// TIA Portal project "OpcUaClient" (V15.1)

(* hardware
DEVICE "S71500/ET200MP-Station_1"  S7-1500 station
   slot 0: "Profilschiene_0"  Rack  6ES7 590-1***0-0AA0
   slot 1: "PLC"  CPU 1513F-1 PN  6ES7 513-1FL02-0AB0  V2.6
      slot 3: "CPU-Display_1"  6ES7591-1AA00-0AA0
*)

// ===== PLC "PLC"  CPU 1513F-1 PN =====

VAR_GLOBAL   // PLC tag table "Standard-Variablentabelle"
   "System_Byte" AT %MB1 : Byte;
   "FirstScan" AT %M1.0 : Bool;
   "DiagStatusUpdate" AT %M1.1 : Bool;
   "AlwaysTRUE" AT %M1.2 : Bool;
   "AlwaysFALSE" AT %M1.3 : Bool;
   "Clock_Byte" AT %MB0 : Byte;
   "Clock_10Hz" AT %M0.0 : Bool;
   "Clock_5Hz" AT %M0.1 : Bool;
   "Clock_2.5Hz" AT %M0.2 : Bool;
   "Clock_2Hz" AT %M0.3 : Bool;
   "Clock_1.25Hz" AT %M0.4 : Bool;
   "Clock_1Hz" AT %M0.5 : Bool;
   "Clock_0.625Hz" AT %M0.6 : Bool;
   "Clock_0.5Hz" AT %M0.7 : Bool;
   "Tag_1" AT %M100.0 : Bool;
   "Tag_2" AT %M300.0 : Bool;
   "Tag_3" AT %M300.1 : Bool;
   "Tag_4" AT %MD310 : DWord;
   "Tag_5" AT %M300.2 : Bool;
   "Tag_6" AT %M200.0 : Bool;
   "Tag_7" AT %M200.2 : Bool;
   "Tag_8" AT %MD210 : DWord;
   "Tag_9" AT %M200.1 : Bool;
   "Tag_10" AT %M600.0 : Bool;
   "Tag_11" AT %M400.0 : Bool;
   "Tag_12" AT %M1000.0 : Bool;
   "Tag_13" AT %M1000.1 : Bool;
   "Tag_14" AT %M1000.2 : Bool;
   "Tag_15" AT %M1000.3 : Bool;
   "Tag_16" AT %M1000.4 : Bool;
   "Tag_17" AT %M1000.5 : Bool;
END_VAR

VAR_GLOBAL CONSTANT   // PLC tag table "Tag table from XML_1"
   "OpcUa_Good" : DWord := 16#00000000;   // Everything is as expected.
   "OpcUa_Uncertain" : DWord := 16#40000000;   // Something unexpected occurred but the results still maybe useable.
   "OpcUa_Bad" : DWord := 16#80000000;   // An error occurred.
   "OpcUa_BadUnexpectedError" : DWord := 16#80010000;   // An unexpected error occurred.
   "OpcUa_BadInternalError" : DWord := 16#80020000;   // An internal error occurred as a result of a programming or configuration error.
   "OpcUa_BadOutOfMemory" : DWord := 16#80030000;   // Not enough memory to complete the operation.
   "OpcUa_BadResourceUnavailable" : DWord := 16#80040000;   // An operating system resource is not available.
   "OpcUa_BadCommunicationError" : DWord := 16#80050000;   // A low level communication error occurred.
   "OpcUa_BadEncodingError" : DWord := 16#80060000;   // Encoding halted because of invalid data in the objects being serialized.
   "OpcUa_BadDecodingError" : DWord := 16#80070000;   // Decoding halted because of invalid data in the stream.
   "OpcUa_BadEncodingLimitsExceeded" : DWord := 16#80080000;   // The message encoding/decoding limits imposed by the stack have been exceeded.
   "OpcUa_BadRequestTooLarge" : DWord := 16#80B80000;   // The request message size exceeds limits set by the server.
   "OpcUa_BadResponseTooLarge" : DWord := 16#80B90000;   // The response message size exceeds limits set by the client.
   "OpcUa_BadUnknownResponse" : DWord := 16#80090000;   // An unrecognized response was received from the server.
   "OpcUa_BadTimeout" : DWord := 16#800A0000;   // The operation timed out.
   "OpcUa_BadServiceUnsupported" : DWord := 16#800B0000;   // The server does not support the requested service.
   "OpcUa_BadShutdown" : DWord := 16#800C0000;   // The operation was cancelled because the application is shutting down.
   "OpcUa_BadServerNotConnected" : DWord := 16#800D0000;   // The operation could not complete because the client is not connected to the server.
   "OpcUa_BadServerHalted" : DWord := 16#800E0000;   // The server has stopped and cannot process any requests.
   "OpcUa_BadNothingToDo" : DWord := 16#800F0000;   // There was nothing to do because the client passed a list of operations with no elements.
   "OpcUa_BadTooManyOperations" : DWord := 16#80100000;   // The request could not be processed because it specified too many operations.
   "OpcUa_BadTooManyMonitoredItems" : DWord := 16#80DB0000;   // The request could not be processed because there are too many monitored items in the subscription.
   "OpcUa_BadDataTypeIdUnknown" : DWord := 16#80110000;   // The extension object cannot be (de)serialized because the data type id is not recognized.
   "OpcUa_BadCertificateInvalid" : DWord := 16#80120000;   // The certificate provided as a parameter is not valid.
   "OpcUa_BadSecurityChecksFailed" : DWord := 16#80130000;   // An error occurred verifying security.
   "OpcUa_BadCertificateTimeInvalid" : DWord := 16#80140000;   // The certificate has expired or is not yet valid.
   "OpcUa_BadCertificateIssuerTimeInvalid" : DWord := 16#80150000;   // An issuer certificate has expired or is not yet valid.
   "OpcUa_BadCertificateHostNameInvalid" : DWord := 16#80160000;   // The HostName used to connect to a server does not match a HostName in the certificate.
   "OpcUa_BadCertificateUriInvalid" : DWord := 16#80170000;   // The URI specified in the ApplicationDescription does not match the URI in the certificate.
   "OpcUa_BadCertificateUseNotAllowed" : DWord := 16#80180000;   // The certificate may not be used for the requested operation.
   "OpcUa_BadCertificateIssuerUseNotAllowed" : DWord := 16#80190000;   // The issuer certificate may not be used for the requested operation.
   "OpcUa_BadCertificateUntrusted" : DWord := 16#801A0000;   // The certificate is not trusted.
   "OpcUa_BadCertificateRevocationUnknown" : DWord := 16#801B0000;   // It was not possible to determine if the certificate has been revoked.
   "OpcUa_BadCertificateIssuerRevocationUnknown" : DWord := 16#801C0000;   // It was not possible to determine if the issuer certificate has been revoked.
   "OpcUa_BadCertificateRevoked" : DWord := 16#801D0000;   // The certificate has been revoked.
   "OpcUa_BadCertificateIssuerRevoked" : DWord := 16#801E0000;   // The issuer certificate has been revoked.
   "OpcUa_BadCertificateChainIncomplete" : DWord := 16#810D0000;   // The certificate chain is incomplete.
   "OpcUa_BadUserAccessDenied" : DWord := 16#801F0000;   // User does not have permission to perform the requested operation.
   "OpcUa_BadIdentityTokenInvalid" : DWord := 16#80200000;   // The user identity token is not valid.
   "OpcUa_BadIdentityTokenRejected" : DWord := 16#80210000;   // The user identity token is valid but the server has rejected it.
   "OpcUa_BadSecureChannelIdInvalid" : DWord := 16#80220000;   // The specified secure channel is no longer valid.
   "OpcUa_BadInvalidTimestamp" : DWord := 16#80230000;   // The timestamp is outside the range allowed by the server.
   "OpcUa_BadNonceInvalid" : DWord := 16#80240000;   // The nonce does appear to be not a random value or it is not the correct length.
   "OpcUa_BadSessionIdInvalid" : DWord := 16#80250000;   // The session id is not valid.
   "OpcUa_BadSessionClosed" : DWord := 16#80260000;   // The session was closed by the client.
   "OpcUa_BadSessionNotActivated" : DWord := 16#80270000;   // The session cannot be used because ActivateSession has not been called.
   "OpcUa_BadSubscriptionIdInvalid" : DWord := 16#80280000;   // The subscription id is not valid.
   "OpcUa_BadRequestHeaderInvalid" : DWord := 16#802A0000;   // The header for the request is missing or invalid.
   "OpcUa_BadTimestampsToReturnInvalid" : DWord := 16#802B0000;   // The timestamps to return parameter is invalid.
   "OpcUa_BadRequestCancelledByClient" : DWord := 16#802C0000;   // The request was cancelled by the client.
   "OpcUa_BadTooManyArguments" : DWord := 16#80E50000;   // Too many arguments were provided.
   "OpcUa_BadLicenseExpired" : DWord := 16#810E0000;   // The server requires a license to operate in general or to perform a service or operation, but existing license is expired.
   "OpcUa_BadLicenseLimitsExceeded" : DWord := 16#810F0000;   // The server has limits on number of allowed operations / objects, based on installed licenses, and these limits where exceeded.
   "OpcUa_BadLicenseNotAvailable" : DWord := 16#81100000;   // The server does not have a license which is required to operate in general or to perform a service or operation.
   "OpcUa_GoodSubscriptionTransferred" : DWord := 16#002D0000;   // The subscription was transferred to another session.
   "OpcUa_GoodCompletesAsynchronously" : DWord := 16#002E0000;   // The processing will complete asynchronously.
   "OpcUa_GoodOverload" : DWord := 16#002F0000;   // Sampling has slowed down due to resource limitations.
   "OpcUa_GoodClamped" : DWord := 16#00300000;   // The value written was accepted but was clamped.
   "OpcUa_BadNoCommunication" : DWord := 16#80310000;   // Communication with the data source is defined, but not established, and there is no last known value available.
   "OpcUa_BadWaitingForInitialData" : DWord := 16#80320000;   // Waiting for the server to obtain values from the underlying data source.
   "OpcUa_BadNodeIdInvalid" : DWord := 16#80330000;   // The syntax of the node id is not valid.
   "OpcUa_BadNodeIdUnknown" : DWord := 16#80340000;   // The node id refers to a node that does not exist in the server address space.
   "OpcUa_BadAttributeIdInvalid" : DWord := 16#80350000;   // The attribute is not supported for the specified Node.
   "OpcUa_BadIndexRangeInvalid" : DWord := 16#80360000;   // The syntax of the index range parameter is invalid.
   "OpcUa_BadIndexRangeNoData" : DWord := 16#80370000;   // No data exists within the range of indexes specified.
   "OpcUa_BadDataEncodingInvalid" : DWord := 16#80380000;   // The data encoding is invalid.
   "OpcUa_BadDataEncodingUnsupported" : DWord := 16#80390000;   // The server does not support the requested data encoding for the node.
   "OpcUa_BadNotReadable" : DWord := 16#803A0000;   // The access level does not allow reading or subscribing to the Node.
   "OpcUa_BadNotWritable" : DWord := 16#803B0000;   // The access level does not allow writing to the Node.
   "OpcUa_BadOutOfRange" : DWord := 16#803C0000;   // The value was out of range.
   "OpcUa_BadNotSupported" : DWord := 16#803D0000;   // The requested operation is not supported.
   "OpcUa_BadNotFound" : DWord := 16#803E0000;   // A requested item was not found or a search operation ended without success.
   "OpcUa_BadObjectDeleted" : DWord := 16#803F0000;   // The object cannot be used because it has been deleted.
   "OpcUa_BadNotImplemented" : DWord := 16#80400000;   // Requested operation is not implemented.
   "OpcUa_BadMonitoringModeInvalid" : DWord := 16#80410000;   // The monitoring mode is invalid.
   "OpcUa_BadMonitoredItemIdInvalid" : DWord := 16#80420000;   // The monitoring item id does not refer to a valid monitored item.
   "OpcUa_BadMonitoredItemFilterInvalid" : DWord := 16#80430000;   // The monitored item filter parameter is not valid.
   "OpcUa_BadMonitoredItemFilterUnsupported" : DWord := 16#80440000;   // The server does not support the requested monitored item filter.
   "OpcUa_BadFilterNotAllowed" : DWord := 16#80450000;   // A monitoring filter cannot be used in combination with the attribute specified.
   "OpcUa_BadStructureMissing" : DWord := 16#80460000;   // A mandatory structured parameter was missing or null.
   "OpcUa_BadEventFilterInvalid" : DWord := 16#80470000;   // The event filter is not valid.
   "OpcUa_BadContentFilterInvalid" : DWord := 16#80480000;   // The content filter is not valid.
   "OpcUa_BadFilterOperatorInvalid" : DWord := 16#80C10000;   // An unregognized operator was provided in a filter.
   "OpcUa_BadFilterOperatorUnsupported" : DWord := 16#80C20000;   // A valid operator was provided, but the server does not provide support for this filter operator.
   "OpcUa_BadFilterOperandCountMismatch" : DWord := 16#80C30000;   // The number of operands provided for the filter operator was less then expected for the operand provided.
   "OpcUa_BadFilterOperandInvalid" : DWord := 16#80490000;   // The operand used in a content filter is not valid.
   "OpcUa_BadFilterElementInvalid" : DWord := 16#80C40000;   // The referenced element is not a valid element in the content filter.
   "OpcUa_BadFilterLiteralInvalid" : DWord := 16#80C50000;   // The referenced literal is not a valid value.
   "OpcUa_BadContinuationPointInvalid" : DWord := 16#804A0000;   // The continuation point provide is longer valid.
   "OpcUa_BadNoContinuationPoints" : DWord := 16#804B0000;   // The operation could not be processed because all continuation points have been allocated.
   "OpcUa_BadReferenceTypeIdInvalid" : DWord := 16#804C0000;   // The operation could not be processed because all continuation points have been allocated.
   "OpcUa_BadBrowseDirectionInvalid" : DWord := 16#804D0000;   // The browse direction is not valid.
   "OpcUa_BadNodeNotInView" : DWord := 16#804E0000;   // The node is not part of the view.
   "OpcUa_BadNumericOverflow" : DWord := 16#81120000;   // The number was not accepted because of a numeric overflow.
   "OpcUa_BadServerUriInvalid" : DWord := 16#804F0000;   // The ServerUri is not a valid URI.
   "OpcUa_BadServerNameMissing" : DWord := 16#80500000;   // No ServerName was specified.
   "OpcUa_BadDiscoveryUrlMissing" : DWord := 16#80510000;   // No DiscoveryUrl was specified.
   "OpcUa_BadSempahoreFileMissing" : DWord := 16#80520000;   // The semaphore file specified by the client is not valid.
   "OpcUa_BadRequestTypeInvalid" : DWord := 16#80530000;   // The security token request type is not valid.
   "OpcUa_BadSecurityModeRejected" : DWord := 16#80540000;   // The security mode does not meet the requirements set by the server.
   "OpcUa_BadSecurityPolicyRejected" : DWord := 16#80550000;   // The security policy does not meet the requirements set by the server.
   "OpcUa_BadTooManySessions" : DWord := 16#80560000;   // The server has reached its maximum number of sessions.
   "OpcUa_BadUserSignatureInvalid" : DWord := 16#80570000;   // The user token signature is missing or invalid.
   "OpcUa_BadApplicationSignatureInvalid" : DWord := 16#80580000;   // The signature generated with the client certificate is missing or invalid.
   "OpcUa_BadNoValidCertificates" : DWord := 16#80590000;   // The client did not provide at least one software certificate that is valid and meets the profile requirements for the server.
   "OpcUa_BadIdentityChangeNotSupported" : DWord := 16#80C60000;   // The server does not support changing the user identity assigned to the session.
   "OpcUa_BadRequestCancelledByRequest" : DWord := 16#805A0000;   // The request was cancelled by the client with the Cancel service.
   "OpcUa_BadParentNodeIdInvalid" : DWord := 16#805B0000;   // The parent node id does not to refer to a valid node.
   "OpcUa_BadReferenceNotAllowed" : DWord := 16#805C0000;   // The reference could not be created because it violates constraints imposed by the data model.
   "OpcUa_BadNodeIdRejected" : DWord := 16#805D0000;   // The requested node id was reject because it was either invalid or server does not allow node ids to be specified by the client.
   "OpcUa_BadNodeIdExists" : DWord := 16#805E0000;   // The requested node id is already used by another node.
   "OpcUa_BadNodeClassInvalid" : DWord := 16#805F0000;   // The node class is not valid.
   "OpcUa_BadBrowseNameInvalid" : DWord := 16#80600000;   // The browse name is invalid.
   "OpcUa_BadBrowseNameDuplicated" : DWord := 16#80610000;   // The browse name is not unique among nodes that share the same relationship with the parent.
   "OpcUa_BadNodeAttributesInvalid" : DWord := 16#80620000;   // The node attributes are not valid for the node class.
   "OpcUa_BadTypeDefinitionInvalid" : DWord := 16#80630000;   // The type definition node id does not reference an appropriate type node.
   "OpcUa_BadSourceNodeIdInvalid" : DWord := 16#80640000;   // The source node id does not reference a valid node.
   "OpcUa_BadTargetNodeIdInvalid" : DWord := 16#80650000;   // The target node id does not reference a valid node.
   "OpcUa_BadDuplicateReferenceNotAllowed" : DWord := 16#80660000;   // The reference type between the nodes is already defined.
   "OpcUa_BadInvalidSelfReference" : DWord := 16#80670000;   // The server does not allow this type of self reference on this node.
   "OpcUa_BadReferenceLocalOnly" : DWord := 16#80680000;   // The reference type is not valid for a reference to a remote server.
   "OpcUa_BadNoDeleteRights" : DWord := 16#80690000;   // The server will not allow the node to be deleted.
   "OpcUa_UncertainReferenceNotDeleted" : DWord := 16#40BC0000;   // The server was not able to delete all target references.
   "OpcUa_BadServerIndexInvalid" : DWord := 16#806A0000;   // The server index is not valid.
   "OpcUa_BadViewIdUnknown" : DWord := 16#806B0000;   // The view id does not refer to a valid view node.
   "OpcUa_BadViewTimestampInvalid" : DWord := 16#80C90000;   // The view timestamp is not available or not supported.
   "OpcUa_BadViewParameterMismatch" : DWord := 16#80CA0000;   // The view parameters are not consistent with each other.
   "OpcUa_BadViewVersionInvalid" : DWord := 16#80CB0000;   // The view version is not available or not supported.
   "OpcUa_UncertainNotAllNodesAvailable" : DWord := 16#40C00000;   // The list of references may not be complete because the underlying system is not available.
   "OpcUa_GoodResultsMayBeIncomplete" : DWord := 16#00BA0000;   // The server should have followed a reference to a node in a remote server but did not. The result set may be incomplete.
   "OpcUa_BadNotTypeDefinition" : DWord := 16#80C80000;   // The provided Nodeid was not a type definition nodeid.
   "OpcUa_UncertainReferenceOutOfServer" : DWord := 16#406C0000;   // One of the references to follow in the relative path references to a node in the address space in another server.
   "OpcUa_BadTooManyMatches" : DWord := 16#806D0000;   // The requested operation has too many matches to return.
   "OpcUa_BadQueryTooComplex" : DWord := 16#806E0000;   // The requested operation requires too many resources in the server.
   "OpcUa_BadNoMatch" : DWord := 16#806F0000;   // The requested operation has no match to return.
   "OpcUa_BadMaxAgeInvalid" : DWord := 16#80700000;   // The max age parameter is invalid.
   "OpcUa_BadSecurityModeInsufficient" : DWord := 16#80E60000;   // The operation is not permitted over the current secure channel.
   "OpcUa_BadHistoryOperationInvalid" : DWord := 16#80710000;   // The history details parameter is not valid.
   "OpcUa_BadHistoryOperationUnsupported" : DWord := 16#80720000;   // The server does not support the requested operation.
   "OpcUa_BadInvalidTimestampArgument" : DWord := 16#80BD0000;   // The defined timestamp to return was invalid.
   "OpcUa_BadWriteNotSupported" : DWord := 16#80730000;   // The server does not support writing the combination of value, status and timestamps provided.
   "OpcUa_BadTypeMismatch" : DWord := 16#80740000;   // The value supplied for the attribute is not of the same type as the attributes value.
   "OpcUa_BadMethodInvalid" : DWord := 16#80750000;   // The method id does not refer to a method for the specified object.
   "OpcUa_BadArgumentsMissing" : DWord := 16#80760000;   // The client did not specify all of the input arguments for the method.
   "OpcUa_BadNotExecutable" : DWord := 16#81110000;   // The executable attribute does not allow the execution of the method.
   "OpcUa_BadTooManySubscriptions" : DWord := 16#80770000;   // The server has reached its maximum number of subscriptions.
   "OpcUa_BadTooManyPublishRequests" : DWord := 16#80780000;   // The server has reached the maximum number of queued publish requests.
   "OpcUa_BadNoSubscription" : DWord := 16#80790000;   // There is no subscription available for this session.
   "OpcUa_BadSequenceNumberUnknown" : DWord := 16#807A0000;   // The sequence number is unknown to the server.
   "OpcUa_BadMessageNotAvailable" : DWord := 16#807B0000;   // The requested notification message is no longer available.
   "OpcUa_BadInsufficientClientProfile" : DWord := 16#807C0000;   // The client of the current session does not support one or more Profiles that are necessary for the subscription.
   "OpcUa_BadStateNotActive" : DWord := 16#80BF0000;   // The sub-state machine is not currently active.
   "OpcUa_BadTcpServerTooBusy" : DWord := 16#807D0000;   // The server cannot process the request because it is too busy.
   "OpcUa_BadTcpMessageTypeInvalid" : DWord := 16#807E0000;   // The type of the message specified in the header invalid.
   "OpcUa_BadTcpSecureChannelUnknown" : DWord := 16#807F0000;   // The SecureChannelId and/or TokenId are not currently in use.
   "OpcUa_BadTcpMessageTooLarge" : DWord := 16#80800000;   // The size of the message specified in the header is too large.
   "OpcUa_BadTcpNotEnoughResources" : DWord := 16#80810000;   // There are not enough resources to process the request.
   "OpcUa_BadTcpInternalError" : DWord := 16#80820000;   // An internal error occurred.
   "OpcUa_BadTcpEndpointUrlInvalid" : DWord := 16#80830000;   // The server does not recognize the QueryString specified.
   "OpcUa_BadRequestInterrupted" : DWord := 16#80840000;   // The request could not be sent because of a network interruption.
   "OpcUa_BadRequestTimeout" : DWord := 16#80850000;   // Timeout occurred while processing the request.
   "OpcUa_BadSecureChannelClosed" : DWord := 16#80860000;   // The secure channel has been closed.
   "OpcUa_BadSecureChannelTokenUnknown" : DWord := 16#80870000;   // The token has expired or is not recognized.
   "OpcUa_BadSequenceNumberInvalid" : DWord := 16#80880000;   // The sequence number is not valid.
   "OpcUa_BadProtocolVersionUnsupported" : DWord := 16#80BE0000;   // The applications do not have compatible protocol versions.
   "OpcUa_BadConfigurationError" : DWord := 16#80890000;   // There is a problem with the configuration that affects the usefulness of the value.
   "OpcUa_BadNotConnected" : DWord := 16#808A0000;   // The variable should receive its value from another variable, but has never been configured to do so.
   "OpcUa_BadDeviceFailure" : DWord := 16#808B0000;   // There has been a failure in the device/data source that generates the value that has affected the value.
   "OpcUa_BadSensorFailure" : DWord := 16#808C0000;   // There has been a failure in the sensor from which the value is derived by the device/data source.
   "OpcUa_BadOutOfService" : DWord := 16#808D0000;   // The source of the data is not operational.
   "OpcUa_BadDeadbandFilterInvalid" : DWord := 16#808E0000;   // The deadband filter is not valid.
   "OpcUa_UncertainNoCommunicationLastUsableValue" : DWord := 16#408F0000;   // Communication to the data source has failed. The variable value is the last value that had a good quality.
   "OpcUa_UncertainLastUsableValue" : DWord := 16#40900000;   // Whatever was updating this value has stopped doing so.
   "OpcUa_UncertainSubstituteValue" : DWord := 16#40910000;   // The value is an operational value that was manually overwritten.
   "OpcUa_UncertainInitialValue" : DWord := 16#40920000;   // The value is an initial value for a variable that normally receives its value from another variable.
   "OpcUa_UncertainSensorNotAccurate" : DWord := 16#40930000;   // The value is at one of the sensor limits.
   "OpcUa_UncertainEngineeringUnitsExceeded" : DWord := 16#40940000;   // The value is outside of the range of values defined for this parameter.
   "OpcUa_UncertainSubNormal" : DWord := 16#40950000;   // The value is derived from multiple sources and has less than the required number of Good sources.
   "OpcUa_GoodLocalOverride" : DWord := 16#00960000;   // The value has been overridden.
   "OpcUa_BadRefreshInProgress" : DWord := 16#80970000;   // This Condition refresh failed, a Condition refresh operation is already in progress.
   "OpcUa_BadConditionAlreadyDisabled" : DWord := 16#80980000;   // This condition has already been disabled.
   "OpcUa_BadConditionAlreadyEnabled" : DWord := 16#80CC0000;   // This condition has already been enabled.
   "OpcUa_BadConditionDisabled" : DWord := 16#80990000;   // Property not available, this condition is disabled.
   "OpcUa_BadEventIdUnknown" : DWord := 16#809A0000;   // The specified event id is not recognized.
   "OpcUa_BadEventNotAcknowledgeable" : DWord := 16#80BB0000;   // The event cannot be acknowledged.
   "OpcUa_BadDialogNotActive" : DWord := 16#80CD0000;   // The dialog condition is not active.
   "OpcUa_BadDialogResponseInvalid" : DWord := 16#80CE0000;   // The response is not valid for the dialog.
   "OpcUa_BadConditionBranchAlreadyAcked" : DWord := 16#80CF0000;   // The condition branch has already been acknowledged.
   "OpcUa_BadConditionBranchAlreadyConfirmed" : DWord := 16#80D00000;   // The condition branch has already been confirmed.
   "OpcUa_BadConditionAlreadyShelved" : DWord := 16#80D10000;   // The condition has already been shelved.
   "OpcUa_BadConditionNotShelved" : DWord := 16#80D20000;   // The condition is not currently shelved.
   "OpcUa_BadShelvingTimeOutOfRange" : DWord := 16#80D30000;   // The shelving time not within an acceptable range.
   "OpcUa_BadNoData" : DWord := 16#809B0000;   // No data exists for the requested time range or event filter.
   "OpcUa_BadBoundNotFound" : DWord := 16#80D70000;   // No data found to provide upper or lower bound value.
   "OpcUa_BadBoundNotSupported" : DWord := 16#80D80000;   // The server cannot retrieve a bound for the variable.
   "OpcUa_BadDataLost" : DWord := 16#809D0000;   // Data is missing due to collection started/stopped/lost.
   "OpcUa_BadDataUnavailable" : DWord := 16#809E0000;   // Expected data is unavailable for the requested time range due to an un-mounted volume, an off-line archive or tape, or similar reason for temporary unavailability.
   "OpcUa_BadEntryExists" : DWord := 16#809F0000;   // The data or event was not successfully inserted because a matching entry exists.
   "OpcUa_BadNoEntryExists" : DWord := 16#80A00000;   // The data or event was not successfully updated because no matching entry exists.
   "OpcUa_BadTimestampNotSupported" : DWord := 16#80A10000;   // The client requested history using a timestamp format the server does not support (i.e requested ServerTimestamp when server only supports SourceTimestamp).
   "OpcUa_GoodEntryInserted" : DWord := 16#00A20000;   // The data or event was successfully inserted into the historical database.
   "OpcUa_GoodEntryReplaced" : DWord := 16#00A30000;   // The data or event field was successfully replaced in the historical database.
   "OpcUa_UncertainDataSubNormal" : DWord := 16#40A40000;   // The value is derived from multiple values and has less than the required number of Good values.
   "OpcUa_GoodNoData" : DWord := 16#00A50000;   // No data exists for the requested time range or event filter.
   "OpcUa_GoodMoreData" : DWord := 16#00A60000;   // The data or event field was successfully replaced in the historical database.
   "OpcUa_BadAggregateListMismatch" : DWord := 16#80D40000;   // The requested number of Aggregates does not match the requested number of NodeIds.
   "OpcUa_BadAggregateNotSupported" : DWord := 16#80D50000;   // The requested Aggregate is not support by the server.
   "OpcUa_BadAggregateInvalidInputs" : DWord := 16#80D60000;   // The aggregate value could not be derived due to invalid data inputs.
   "OpcUa_BadAggregateConfigurationRejected" : DWord := 16#80DA0000;   // The aggregate configuration is not valid for specified node.
   "OpcUa_GoodDataIgnored" : DWord := 16#00D90000;   // The request pecifies fields which are not valid for the EventType or cannot be saved by the historian.
   "OpcUa_BadRequestNotAllowed" : DWord := 16#80E40000;   // The request was rejected by the server because it did not meet the criteria set by the server.
   "OpcUa_BadRequestNotComplete" : DWord := 16#81130000;   // The request has not been processed by the server yet.
   "OpcUa_GoodEdited" : DWord := 16#00DC0000;   // The value does not come from the real source and has been edited by the server.
   "OpcUa_GoodPostActionFailed" : DWord := 16#00DD0000;   // There was an error in execution of these post-actions.
   "OpcUa_UncertainDominantValueChanged" : DWord := 16#40DE0000;   // The related EngineeringUnit has been changed but the Variable Value is still provided based on the previous unit.
   "OpcUa_GoodDependentValueChanged" : DWord := 16#00E00000;   // A dependent value has been changed but the change has not been applied to the device.
   "OpcUa_BadDominantValueChanged" : DWord := 16#80E10000;   // The related EngineeringUnit has been changed but this change has not been applied to the device. The Variable Value is still dependent on the previous unit but its status is currently Bad.
   "OpcUa_UncertainDependentValueChanged" : DWord := 16#40E20000;   // A dependent value has been changed but the change has not been applied to the device. The quality of the dominant variable is uncertain.
   "OpcUa_BadDependentValueChanged" : DWord := 16#80E30000;   // A dependent value has been changed but the change has not been applied to the device. The quality of the dominant variable is Bad.
   "OpcUa_GoodCommunicationEvent" : DWord := 16#00A70000;   // The communication layer has raised an event.
   "OpcUa_GoodShutdownEvent" : DWord := 16#00A80000;   // The system is shutting down.
   "OpcUa_GoodCallAgain" : DWord := 16#00A90000;   // The operation is not finished and needs to be called again.
   "OpcUa_GoodNonCriticalTimeout" : DWord := 16#00AA0000;   // A non-critical timeout occurred.
   "OpcUa_BadInvalidArgument" : DWord := 16#80AB0000;   // One or more arguments are invalid.
   "OpcUa_BadConnectionRejected" : DWord := 16#80AC0000;   // Could not establish a network connection to remote server.
   "OpcUa_BadDisconnect" : DWord := 16#80AD0000;   // The server has disconnected from the client.
   "OpcUa_BadConnectionClosed" : DWord := 16#80AE0000;   // The network connection has been closed.
   "OpcUa_BadInvalidState" : DWord := 16#80AF0000;   // The operation cannot be completed because the object is closed, uninitialized or in some other invalid state.
   "OpcUa_BadEndOfStream" : DWord := 16#80B00000;   // Cannot move beyond end of the stream.
   "OpcUa_BadNoDataAvailable" : DWord := 16#80B10000;   // No data is currently available for reading from a non-blocking stream.
   "OpcUa_BadWaitingForResponse" : DWord := 16#80B20000;   // The asynchronous operation is waiting for a response.
   "OpcUa_BadOperationAbandoned" : DWord := 16#80B30000;   // The asynchronous operation was abandoned by the caller.
   "OpcUa_BadExpectedStreamToBlock" : DWord := 16#80B40000;   // The stream did not return all data requested (possibly because it is a non-blocking stream).
   "OpcUa_BadWouldBlock" : DWord := 16#80B50000;   // Non blocking behaviour is required and the operation would block.
   "OpcUa_BadSyntaxError" : DWord := 16#80B60000;   // A value had an invalid syntax.
   "OpcUa_BadMaxConnectionsReached" : DWord := 16#80B70000;   // The operation could not be finished because all available connections are in use.
END_VAR

TYPE "MyMethodInType"
   STRUCT
      "Afotek-ID" : UInt;
   END_STRUCT;
END_TYPE

TYPE "MyMethodOutType"
   STRUCT
      "Afotek-ID" : UInt;
      "Erfal-ID" : ULInt;
      Beizzeit : UInt;
      Spuelen1 : UInt;
      "VE-Spuelen1" : UInt;
      Passivierung : UInt;
      "VE-Spuelen2" : UInt;
      "HWT-Time" : UInt;
      "HWT-Cooltime" : UInt;
      "Pulver-PGNO" : UInt;
      "Pulver-Color" : String;
      "PEO-Temperatur" : UInt;
      "PEO-Time" : UInt;
      "PEO-Cooltime" : UInt;
   END_STRUCT;
END_TYPE

// folder: Siemens OPC Client

TYPE "connectionParameterType"
   STRUCT
      ConnectInfo : OPC_UA_SessionConnectInfo;
      ConnectionHdl : DWord;
      ServerEndpointUrl : String[254] := 'opc.tcp://192.168.0.2:4840';
   END_STRUCT;
   // ConnectInfo.SessionName := WSTRING#'OPC UA Connection_1';
   // ConnectInfo.ApplicationName := WSTRING#'';
   // ConnectInfo.SecurityMsgMode := 1;
   // ConnectInfo.SecurityPolicy := 1;
   // ConnectInfo.ServerUri := '';
   // ConnectInfo.CheckServerCertificate := False;
   // ConnectInfo.TransportProfile := 1;
   // ConnectInfo.UserIdentityTokenType := 0;
   // ConnectInfo.CertificateID := 0;
   // ConnectInfo.SessionTimeout := T#30S;
   // ConnectInfo.MonitorConnection := T#5S;
   // ConnectInfo.LocaleIDs[0] := 'en-US';
   // ConnectInfo.LocaleIDs[1] := '';
   // ConnectInfo.LocaleIDs[2] := '';
   // ConnectInfo.LocaleIDs[3] := '';
   // ConnectInfo.LocaleIDs[4] := '';
END_TYPE

TYPE "methodListType"
   STRUCT
      MethodCount : UInt;
      ObjectNodes : Array[0..0] of OPC_UA_NodeId;
      MethodNodes : Array[0..0] of OPC_UA_NodeId;
      MethodHdls : Array[0..0] of DWord;
   END_STRUCT;
   // ObjectNodes[0].NamespaceIndex := 0;
   // ObjectNodes[0].Identifier := WSTRING#'"OPCMethodSetMachineTime_DB"';
   // ObjectNodes[0].IdentifierType := 1;
   // MethodNodes[0].NamespaceIndex := 0;
   // MethodNodes[0].Identifier := WSTRING#'"OPCMethodSetMachineTime_DB".Method';
   // MethodNodes[0].IdentifierType := 1;
END_TYPE

TYPE "namespaceType"
   STRUCT
      NamespaceURIs : Array[0..0] of WString;
      ServerNamespaceIndexes : Array[0..0] of UInt;
      NamespaceStatusList : Array[0..0] of DWord;
      NamespaceCount : UInt;
   END_STRUCT;
   // NamespaceURIs[0] := WSTRING#'http://www.siemens.com/simatic-s7-opcua';
END_TYPE

TYPE "readWriteListType"
   STRUCT
      NodeCount : UInt;
   END_STRUCT;
END_TYPE

// folder: SystemDataTypeFolder

TYPE "Python.Methodenliste.getData.Inputs"
   STRUCT
      Element_1 : ULInt;
   END_STRUCT;
END_TYPE

TYPE "Python.Methodenliste.getData.Outputs"
   STRUCT
      Element_1 : ULInt;
      Element_2 : ULInt;
   END_STRUCT;
END_TYPE

// folder: (top level)

DATA_BLOCK "Main_Safety_RTG1_DB"   // DB3, F_DB
{ S7_Optimized_Access := 'TRUE' }
NAME : FUSI
VERSION : 0.1
// stored: InstanceOfName Main_Safety_RTG1
"Main_Safety_RTG1"
BEGIN
END_DATA_BLOCK

// folder: OPC UA/Client

DATA_BLOCK "Clients_DB"   // DB8
{ S7_Optimized_Access := 'TRUE' }
VERSION : 0.1
// stored: InstanceOfName Clients
"Clients"
BEGIN
END_DATA_BLOCK

// folder: OPC UA/Client/Siemens Client

DATA_BLOCK "Python_Configuration"   // DB1
{ S7_Optimized_Access := 'TRUE' }
VERSION : 0.1
   VAR
      Connection : Struct
         ConnectInfo : OPC_UA_SessionConnectInfo;
         ConnectionHdl : DWord;
         ServerEndpointUrl : String[254] := 'opc.tcp://192.168.10.202:4840';
      END_STRUCT;
      Namespaces : Struct
         NamespaceURIs : Array[0..0] of WString;
         ServerNamespaceIndexes : Array[0..0] of UInt;
         NamespaceStatusList : Array[0..0] of DWord;
         NamespaceCount : UInt := 1;
      END_STRUCT;
      MethodLists : Struct
         Methodenliste : Struct
            MethodCount : UInt := 1;
            ObjectNodes : Array[0..0] of OPC_UA_NodeId;
            MethodNodes : Array[0..0] of OPC_UA_NodeId;
            MethodHdls : Array[0..0] of DWord;
         END_STRUCT;
      END_STRUCT;
   END_VAR
BEGIN
   MethodLists.Methodenliste.MethodNodes[0].NamespaceIndex := 0;
   MethodLists.Methodenliste.MethodNodes[0].IdentifierType := 0;
   MethodLists.Methodenliste.MethodNodes[0].Identifier := WSTRING#'4';
   MethodLists.Methodenliste.ObjectNodes[0].NamespaceIndex := 0;
   MethodLists.Methodenliste.ObjectNodes[0].IdentifierType := 0;
   MethodLists.Methodenliste.ObjectNodes[0].Identifier := WSTRING#'3';
   Connection.ConnectInfo.SessionName := WSTRING#'Python';
   Connection.ConnectInfo.ApplicationName := WSTRING#'';
   Connection.ConnectInfo.SecurityMsgMode := 1;
   Connection.ConnectInfo.SecurityPolicy := 1;
   Connection.ConnectInfo.ServerUri := '';
   Connection.ConnectInfo.CheckServerCertificate := False;
   Connection.ConnectInfo.TransportProfile := 1;
   Connection.ConnectInfo.UserIdentityTokenType := 0;
   Connection.ConnectInfo.CertificateID := 0;
   Connection.ConnectInfo.SessionTimeout := T#30S;
   Connection.ConnectInfo.MonitorConnection := T#5S;
   Connection.ConnectInfo.LocaleIDs[0] := 'de-DE';
   Connection.ConnectInfo.LocaleIDs[1] := '';
   Connection.ConnectInfo.LocaleIDs[2] := '';
   Connection.ConnectInfo.LocaleIDs[3] := '';
   Connection.ConnectInfo.LocaleIDs[4] := '';
   Namespaces.NamespaceURIs[0] := WSTRING#'PythonOpcUaServer/namespace/';
END_DATA_BLOCK

DATA_BLOCK "Python_Data"   // DB2
{ S7_Optimized_Access := 'TRUE' }
VERSION : 0.1
   VAR
      Methodenliste : Struct
         MethodStatusList : Array[0..0] of DWord;
         MethodResultList : Array[0..0] of DWord;
         getData : Struct   // getData
            Inputs : "Python.Methodenliste.getData.Inputs";   // InputArguments
            Outputs : "Python.Methodenliste.getData.Outputs";   // OutputArguments
         END_STRUCT;
      END_STRUCT;
   END_VAR
BEGIN
END_DATA_BLOCK

// folder: (top level)

FUNCTION_BLOCK "Main_Safety_RTG1"   // FB1, F_FBD
{ S7_Optimized_Access := 'TRUE' }
VERSION : 0.1
BEGIN
END_FUNCTION_BLOCK

ORGANIZATION_BLOCK "Main"   // OB1, LAD, ProgramCycle
TITLE = "Main Program Sweep (Cycle)"
{ S7_Optimized_Access := 'TRUE' }
VERSION : 0.1
   VAR_INPUT
      Initial_Call : Bool;   // Initial call of this OB
      Remanence : Bool;   // =True, if remanent data are available
   END_VAR
   VAR_TEMP
      tRET_VAL : Word;
   END_VAR
BEGIN

REGION Network 1
   // Test: IO
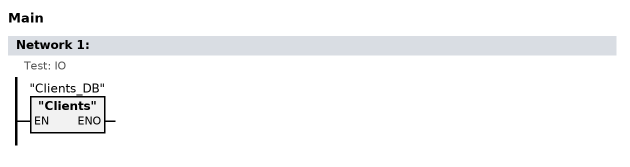
   RUNG wire#powerrail
      "Clients_DB"()
   END_RUNG
   // the same network as SCL:
   "Clients_DB"();   // "Clients"
END_REGION
END_ORGANIZATION_BLOCK

// folder: OPC UA/Client

FUNCTION_BLOCK "Clients"   // FB5, LAD
{ S7_Optimized_Access := 'TRUE' }
VERSION : 0.1
   VAR
      connected : Bool;
      done : Bool;
      busy : Bool;
      error : Bool;
      errorid : Int;
      status : DWord;
      flanke : Bool;
      old_error : Int;
      old_status : DWord;
      OpcUaClient_Instance : "OpcUaClient";
   END_VAR
   VAR_TEMP
      url : String;
   END_VAR
   VAR_TEMP   // added for the SCL form of the ladder/FBD networks
      _w1 : Bool;
   END_VAR
BEGIN

REGION Network 1
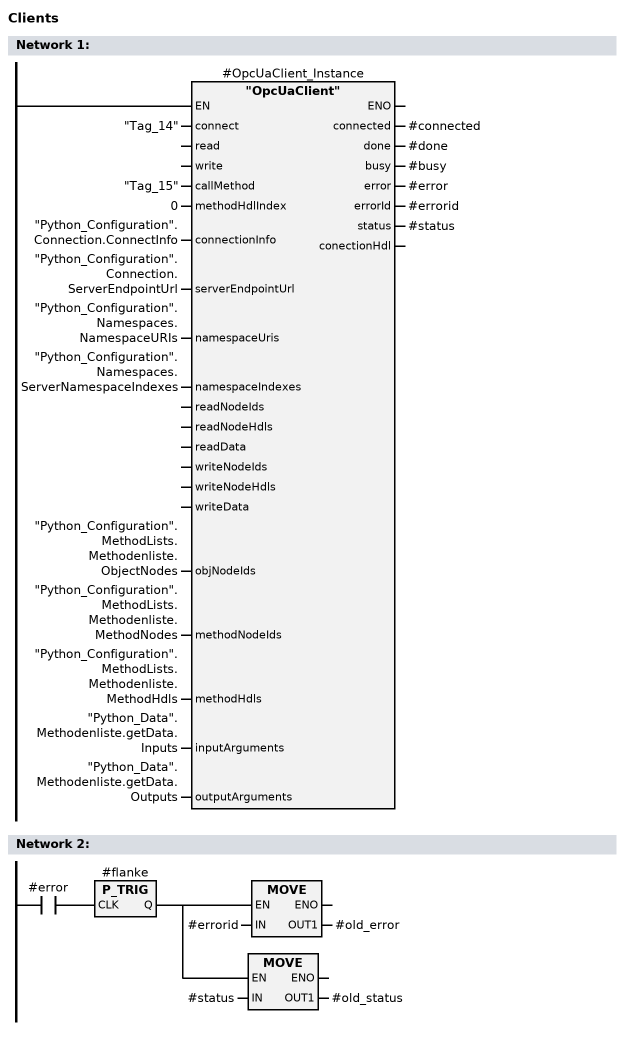
   // no checked SCL form for this network; see the picture
END_REGION

REGION Network 2
   RUNG wire#powerrail
      Contact( #error )
      P_Trig( #flanke )
      wire#w1
      Move(in := #errorid, out1 => #old_error)
   END_RUNG
   RUNG wire#w1
      Move(in := #status, out1 => #old_status)
   END_RUNG
   // the same network as SCL:
   #_w1 := #error AND NOT #flanke;   // rising edge
   #flanke := #error;
   IF #_w1 THEN
       #old_error := #errorid;
       #old_status := #status;
   END_IF;
END_REGION
END_FUNCTION_BLOCK

// folder: OPC UA/Client/Siemens Client

FUNCTION_BLOCK "OpcUaClient"   // FB8, SCL
TITLE = OpcUaClient
{ S7_Optimized_Access := 'TRUE' }
AUTHOR : SiemensAG
VERSION : 1.0
// OPC UA-Client-Wrapper
   VAR_INPUT
      connect : Bool;
      read : Bool;
      write : Bool;
      callMethod : Bool;
      methodHdlIndex : DInt;
      connectionInfo : OPC_UA_SessionConnectInfo;
      serverEndpointUrl : String;
   END_VAR
   VAR_OUTPUT
      connected : Bool;
      done : Bool;
      busy : Bool;
      error : Bool;
      errorId : Int;
      status : DWord;
      conectionHdl : DWord;
   END_VAR
   VAR_IN_OUT
      namespaceUris : Variant;
      namespaceIndexes : Variant;
      readNodeIds : Variant;
      readNodeHdls : Variant;
      readData : Variant;
      writeNodeIds : Variant;
      writeNodeHdls : Variant;
      writeData : Variant;
      objNodeIds : Variant;
      methodNodeIds : Variant;
      methodHdls : Variant;
      inputArguments : Variant;
      outputArguments : Variant;
   END_VAR
   VAR
      instOpcUaConnect : OPC_UA_Connect;
      instOpcUaConnectionGetStatus : OPC_UA_ConnectionGetStatus;
      instOpcUaNamespaceGIL : OPC_UA_NamespaceGetIndexList;
      InstOpcUaGHLRead : OPC_UA_NodeGetHandleList;
      instOpcUaGHLWrite : OPC_UA_NodeGetHandleList;
      instOpcUaGHLMethods : OPC_UA_MethodGetHandleList;
      InstOpcUaRHLRead : OPC_UA_NodeReleaseHandleList;
      instOpcUaRHLWrite : OPC_UA_NodeReleaseHandleList;
      instOpcUaRHLMethods : OPC_UA_MethodReleaseHandleList;
      instOpcUaReadList : OPC_UA_ReadList;
      instOpcUaWriteList : OPC_UA_WriteList;
      instOpcUaMethodCall : OPC_UA_MethodCall;
      instOpcUaDisconnect : OPC_UA_Disconnect;
      instConnRTrig : R_TRIG;
      instDisconRTrig : R_TRIG;
      instReconTrigger : R_TRIG;
      instNGILTrigger : R_TRIG;
      instReadTrigger : R_TRIG;
      instWriteTrigger : R_TRIG;
      instMethodCallTrigger : R_TRIG;
      instClearConnTrig : R_TRIG;
      statCase : Int;
      statDone : Bool;
      statConnected : Bool;
      statBusy : Bool;
      statError : Bool;
      statErrorId : Int;
      statStatus : DWord;
      statOpcUaRequests : Struct
         Connect : Bool;
         ConGS : Bool;
         NGIL : Bool;
         GHLRead : Bool;
         GHLMethods : Bool;
         GHLWrite : Bool;
         Read : Bool;
         Write : Bool;
         MethodCall : Bool;
         RHLRead : Bool;
         RHLWrite : Bool;
         RHLMethods : Bool;
         Disconnect : Bool;
      END_STRUCT;
      statRHLTrigger : Bool;
      statConnectCount : Int;
      statNamespaceIndexesSet : Bool;
      statNamespaceRegCount : Int;
      statRegisteredRead : Bool;
      statRegisterCountRead : Int;
      statRegisteredWrite : Bool;
      statRegisterCountWrite : Int;
      statRegisteredMethods : Bool;
      statRegisterCountMethod : Int;
      statReadCount : Int;
      statWriteCount : Int;
      statMethodCallCount : DWord;
      statMethodResult : DWord;
      statMethodHdl : DWord;
      statMethodHdlId : DInt;
      statConnectionHdl : DWord;
      instCycDiag : TON_TIME;
      statCycDiagTrigger : Bool;
      statOpcUaReadTimeStamps : Array[0..299] of LDT;
      statSerializeMethodHdls : Array[0..1199] of Byte;
      statOpcUaStatusLists : Struct
         MethodRHL : Array[0..299] of DWord;
         MethodGHL : Array[0..299] of DWord;
         WriteRHL : Array[0..299] of DWord;
         WriteList : Array[0..299] of DWord;
         WriteGHL : Array[0..299] of DWord;
         ReadRHL : Array[0..299] of DWord;
         ReadList : Array[0..299] of DWord;
         ReadGHL : Array[0..299] of DWord;
         NamespaceGIL : Array[0..299] of DWord;
      END_STRUCT;
   END_VAR
   VAR_TEMP
      tempConnectTrigger : Bool;
      tempDisconnectTrigger : Bool;
      tempIndex : Int;
      tempReadTrigger : Bool;
      tempWriteTrigger : Bool;
      tempMethodCallTrigger : Bool;
      tempRetVal : Int;
      tempCycDiag : Bool;
      tempReconnectTrigger : Bool;
      tempRHLTrigger : Bool;
   END_VAR
   VAR CONSTANT
      CASE_CONNECT : Int := 0;
      CASE_NAMESPACE_GET_INDEX_LIST : Int := 1;
      CASE_CONNECTION_GET_STATUS : Int := 2;
      CASE_NODE_GET_HANDLE_LIST : Int := 3;
      CASE_CONNECTED : Int := 4;
      UACS_CONNECTED : UDInt := 0;
      UASS_RUNNING : UDInt := 0;
      UASL_GOOD : UDInt := 16#0000_00FF;
      STATUS_SESSION_CLEANEDUP : DWord := 16#A000_0105;
      STATUS_BUSY : Word := 16#7001;
      STATUS_SERVER_NOT_CONNECTED : DWord := 16#800D_0000;
      STATUS_BAD_CONNECTION_CLOSED : DWord := 16#80AE_0000;
      STATUS_IDLE : Word := 16#7000;
      STATUS_NOT_REGISTERED : Word := 16#80FF;
      STATUS_DONE : Word := 16#0000;
      CYC_TIME_GCS : Time := T#5S;
      OPC_UA_FUNCTIONS_TIMEOUT : Time := T#10S;
      ERR_ID_GOOD : SInt := 0;
      ERR_ID_CON : SInt := 1;
      ERR_ID_CON_GS_STATUS : SInt := 10;
      ERR_ID_CON_GS_CSTATE : SInt := 11;
      ERR_ID_CON_GS_SSTATE : SInt := 12;
      ERR_ID_CON_GS_SLVL : SInt := 13;
      ERR_ID_NGIL : SInt := 2;
      ERR_ID_R_GHL : SInt := 31;
      ERR_ID_W_GHL : SInt := 32;
      ERR_ID_M_GHL : SInt := 33;
      ERR_ID_RL : SInt := 4;
      ERR_ID_WL : SInt := 5;
      ERR_ID_MC : SInt := 6;
      ERR_ID_R_RHL : SInt := 71;
      ERR_ID_W_RHL : SInt := 72;
      ERR_ID_M_RHL : SInt := 73;
      ERR_ID_DISCON : SInt := 8;
   END_VAR
BEGIN
   //=============================================================================
   // Siemens AG (c)Copyright (2019)
   //-----------------------------------------------------------------------------
   // Library: -
   // Tested with: CPU 1513-1 PN;  FW 2.6
   // Engineering: TIA Portal (V15.1)
   // Restrictions: -
   // Requirements: OPC UA Client activated, Fimware V2.6; Set PLC time
   // Functionality: Encapsulates OPC UA client blocks for read, write and method
   //                call including connection handling and diagnosis
   //-----------------------------------------------------------------------------
   // Change log table:
   // Version    Date         Expert in charge           Changes applied
   // 01.00.00   01.02.2019   Siemens SUP Applications   First released version
   //=============================================================================


   //State machine
   CASE #statCase OF
     #CASE_CONNECT:
       REGION Connection Handling
         //initialize FB
         IF NOT #connect THEN
           #statError := FALSE;
           #statBusy := FALSE;
           #statDone := FALSE;
           #statConnected := FALSE;
           #statErrorId := #ERR_ID_GOOD;
           #statStatus := #STATUS_DONE;
         END_IF;

         //Rising Edge detection of connect
         #instConnRTrig(CLK := #connect,
                        Q => #tempConnectTrigger);

         #instReconTrigger(CLK := #connect
                           AND NOT #statConnected
                           AND (#statStatus = #STATUS_SESSION_CLEANEDUP OR #statStatus = #STATUS_BAD_CONNECTION_CLOSED),
                           Q => #tempReconnectTrigger);

         //If Connect requested, start connection establishment
         //---------CONNECT HANDLING-------------
         //--------------------------------------
         IF #tempConnectTrigger OR #tempReconnectTrigger THEN
           IF #statConnectionHdl = 16#0 THEN
             // no connectionHdl is used -> ready to connect
             #statOpcUaRequests.Connect := TRUE;
             // set FB outputs
             #statBusy := TRUE;
             #statStatus := #STATUS_BUSY;
           ELSE
             //connectionHdl might be defect, first delete connectionHdl
             //-> not ready to connect
             #statOpcUaRequests.Disconnect := TRUE;
             //set FB Outputs
             #statBusy := TRUE;
             #statStatus := #STATUS_BUSY;
           END_IF;
         ELSE
           IF #instOpcUaDisconnect.Error OR #instOpcUaDisconnect.Done THEN
             //possibly open connection handle is not available or is disconnected
             //-> ready to connect
             #statOpcUaRequests.Disconnect := FALSE;
             #statOpcUaRequests.Connect := TRUE;
             #statConnectionHdl := 0;
           ELSE
             //nothing done by OPC UA Disconnect block -> Not ready to connect
             #statOpcUaRequests.Connect := FALSE;
           END_IF;
         END_IF;

         //Error at connection establishment
         IF #instOpcUaConnect.Error THEN
           #statError := TRUE;
           #statDone := FALSE;
           #statConnected := FALSE;
           #statErrorId := #ERR_ID_CON;
           #statStatus := #instOpcUaConnect.Status;
         END_IF;

         //Connection establishment was successful
         IF #instOpcUaConnect.Done THEN
           #statConnected := TRUE;
           #statError := FALSE;
           #statErrorId := #ERR_ID_GOOD;
           #statConnectCount += 1;
           #statCase := #CASE_NAMESPACE_GET_INDEX_LIST;
         END_IF;

       END_REGION

     #CASE_NAMESPACE_GET_INDEX_LIST:
       REGION Handle Namespaces
         //Request Namespace get Indexlist
         #statOpcUaRequests.NGIL := TRUE;
         #statStatus := #STATUS_BUSY;

         // Get Index List was not successful
         IF #instOpcUaNamespaceGIL.Error THEN
           //--> Call ConnectionGetStatus if Status = "16#800D0000"
           IF #instOpcUaNamespaceGIL.Status = #STATUS_SERVER_NOT_CONNECTED THEN
             #statCase := #CASE_CONNECTION_GET_STATUS;
           ELSE
             #statCase := #CASE_CONNECT;
           END_IF;
           #statOpcUaRequests.NGIL := FALSE;
           // => OUT
           #statError := TRUE;
           #statBusy := FALSE;
           #statStatus := #instOpcUaNamespaceGIL.Status;
           #statErrorId := #ERR_ID_NGIL;
         END_IF;

         //Get Index List was successful
         IF #instOpcUaNamespaceGIL.Done THEN
           //Check StatusList
           FOR #tempIndex := 0 TO UDINT_TO_INT(CountOfElements(#namespaceUris) - 1) DO
             IF #statOpcUaStatusLists.#NamespaceGIL[#tempIndex] <> 16#0 THEN
               #statOpcUaRequests.NGIL := FALSE;
               // => OUT
               #statError := TRUE;
               #statStatus := #statOpcUaStatusLists.NamespaceGIL[#tempIndex];
               #statErrorId := #ERR_ID_NGIL;
               #statCase := #CASE_CONNECT;
               EXIT;
             END_IF;
           END_FOR;
           #statOpcUaRequests.NGIL := FALSE;
           IF NOT #statError THEN
             //Count up statNamespaceGetIndexCount
             #statNamespaceRegCount += 1;
             //statNamespaceIndexesSet
             #statNamespaceIndexesSet := TRUE;
             // => OUT
             #statError := FALSE;
             #statErrorId := #ERR_ID_GOOD;
             //Next Step
             #statCase := #CASE_NODE_GET_HANDLE_LIST;
           ELSE
             #statCase := #CASE_CONNECTION_GET_STATUS;
           END_IF;
         END_IF;
       END_REGION

     #CASE_NODE_GET_HANDLE_LIST:
       REGION Handle NodeId lists
         //Trigger NodeHandleList SFBs
         IF NOT #statRegisteredWrite AND #writeNodeIds <> NULL AND #writeNodeHdls <> NULL THEN
           #statOpcUaRequests.GHLWrite := TRUE;
           #statStatus := #STATUS_BUSY;
         ELSE
           IF NOT #statRegisteredRead AND #readNodeIds <> NULL AND #readNodeHdls <> NULL THEN
             #statOpcUaRequests.GHLRead := TRUE;
             #statStatus := #STATUS_BUSY;
           ELSE
             IF NOT #statRegisteredMethods AND #methodNodeIds <> NULL AND #methodHdls <> NULL AND #objNodeIds <> NULL THEN
               #statOpcUaRequests.GHLMethods := TRUE;
               #statStatus := #STATUS_BUSY;
             ELSE
               #statCase := #CASE_CONNECTED;
               #statBusy := FALSE;
               #statStatus := #STATUS_IDLE;
             END_IF;
           END_IF;
         END_IF;

         REGION Handle ReadList
           //Read Node Get Handle List was not successful
           IF #InstOpcUaGHLRead.Error THEN
             //--> Call ConnectionGetStatus if Status = "16#800D0000"
             IF #InstOpcUaGHLRead.Status = #STATUS_SERVER_NOT_CONNECTED THEN
               #statCase := #CASE_CONNECTION_GET_STATUS;
             ELSE
               //#statCase := #CASE_CONNECT;
               #statCase := #CASE_CONNECTED;
             END_IF;
             #statOpcUaRequests.GHLRead := FALSE;
             // => OUT
             #statError := TRUE;
             #statStatus := #InstOpcUaGHLRead.Status;
             #statErrorId := #ERR_ID_R_GHL;
           END_IF;

           //Read Node Get Handle List was successful
           IF #InstOpcUaGHLRead.Done THEN
             //Check StatusList
             FOR #tempIndex := 0 TO UDINT_TO_INT(CountOfElements(#readNodeIds) - 1) DO
               IF #statOpcUaStatusLists.#ReadGHL[#tempIndex] <> 16#0 THEN
                 // => OUT
                 #statBusy := FALSE;
                 #statError := TRUE;
                 #statStatus := #statOpcUaStatusLists.#ReadGHL[#tempIndex];
                 #statErrorId := #ERR_ID_R_GHL;
                 //#statCase := #CASE_CONNECT;
                 EXIT;
               END_IF;
             END_FOR;
             #statOpcUaRequests.GHLRead := FALSE;
             // Count up statRegisterCount
             #statRegisterCountRead += 1;
             // Nodes are registered
             #statRegisteredRead := TRUE;
             IF NOT #statError THEN
               // => OUT
               #statError := FALSE;
               #statErrorId := #ERR_ID_GOOD;
             END_IF;
           END_IF;
         END_REGION
         REGION Handle Write List
           //Write Node Get Handle List was not successful
           IF #instOpcUaGHLWrite.Error THEN
             //--> Call ConnectionGetStatus if Status = "16#800D0000"
             IF #instOpcUaGHLWrite.Status = #STATUS_SERVER_NOT_CONNECTED THEN
               #statCase := #CASE_CONNECTION_GET_STATUS;
             ELSE
               //#statCase := #CASE_CONNECT;
               #statCase := #CASE_CONNECTED;
             END_IF;
             #statOpcUaRequests.GHLWrite := FALSE;
             // => OUT
             #statError := TRUE;
             #statStatus := #instOpcUaGHLWrite.Status;
             #statErrorId := #ERR_ID_W_GHL;
           END_IF;

           //Write Node Get Handle List was successful
           IF #instOpcUaGHLWrite.Done THEN
             //Check StatusList
             FOR #tempIndex := 0 TO UDINT_TO_INT(CountOfElements(#writeNodeIds) - 1) DO
               IF #statOpcUaStatusLists.#WriteGHL[#tempIndex] <> 16#0 THEN
                 // => OUT
                 #statBusy := FALSE;
                 #statError := TRUE;
                 #statStatus := #statOpcUaStatusLists.#WriteGHL[#tempIndex];
                 #statErrorId := #ERR_ID_W_GHL;
                 //#statCase := #CASE_CONNECT;
                 EXIT;
               END_IF;
             END_FOR;
             #statOpcUaRequests.GHLWrite := FALSE;
             // Count up statRegisterCount
             #statRegisterCountWrite += 1;
             // Nodes are registered
             #statRegisteredWrite := TRUE;
             IF NOT #statError THEN
               // => OUT
               #statError := FALSE;
               #statErrorId := #ERR_ID_GOOD;
             END_IF;
           END_IF;
         END_REGION

         REGION Handle MethodList
           //Method Get HandleList was not successful
           IF #instOpcUaGHLMethods.Error THEN
             //--> Call ConnectionGetStatus if Status = "16#800D0000"
             IF #instOpcUaGHLMethods.Status = #STATUS_SERVER_NOT_CONNECTED THEN
               #statCase := #CASE_CONNECTION_GET_STATUS;
             ELSE
               //#statCase := #CASE_CONNECT;
               #statCase := #CASE_CONNECTED;
             END_IF;
             #statOpcUaRequests.GHLMethods := FALSE;
             // => OUT
             #statError := TRUE;
             #statStatus := #instOpcUaGHLMethods.Status;
             #statErrorId := #ERR_ID_M_GHL;
           END_IF;

           //Method Get Handle List was successful
           IF #instOpcUaGHLMethods.Done THEN
             //Check StatusList
             FOR #tempIndex := 0 TO UDINT_TO_INT(CountOfElements(#methodNodeIds) - 1) DO
               IF #statOpcUaStatusLists.#MethodGHL[#tempIndex] <> 16#0 THEN
                 // => OUT
                 #statBusy := FALSE;
                 #statError := TRUE;
                 #statStatus := #statOpcUaStatusLists.#MethodGHL[#tempIndex];
                 #statErrorId := #ERR_ID_M_GHL;
                 //#statCase := #CASE_CONNECT;
                 EXIT;
               END_IF;
             END_FOR;
             #statOpcUaRequests.GHLMethods := FALSE;
             // Count up statRegisterCount
             #statRegisterCountMethod += 1;
             // Nodes are registered
             #statRegisteredMethods := TRUE;
             IF NOT #statError THEN
               // => OUT
               #statError := FALSE;
               #statErrorId := #ERR_ID_GOOD;
             END_IF;
           END_IF;
         END_REGION

       END_REGION

     #CASE_CONNECTED:

       REGION Command and Idle
         //Idle as long as no Command was triggered
         IF NOT #statBusy AND NOT #read AND NOT #write AND NOT #callMethod THEN
           #statDone := FALSE;
           #statError := FALSE;
           #statErrorId := #ERR_ID_GOOD;
           #statStatus := #STATUS_IDLE;
         END_IF;
         //OPC_UA_GetStatus function is called cyclically, so the connection is monitored
         #instCycDiag(IN := NOT #statCycDiagTrigger,
                      PT := #CYC_TIME_GCS,
                      Q => #tempCycDiag);
         #statCycDiagTrigger := FALSE;
         IF #tempCycDiag AND NOT #statRHLTrigger THEN
           #statCase := #CASE_CONNECTION_GET_STATUS;
           #statCycDiagTrigger := TRUE;
         END_IF;

         REGION Read
           //Trigger
           IF #statRegisteredRead THEN
             #instReadTrigger(CLK := #read,
                              Q => #tempReadTrigger);
           ELSE
             IF #read THEN
               #statError := TRUE;
               #statErrorId := #ERR_ID_RL;
               #statStatus := #STATUS_NOT_REGISTERED; //Error no ReadList is registerd Request denied
             ELSE
               #statError := FALSE;
               #statErrorId := #ERR_ID_GOOD;
               #statStatus := #STATUS_IDLE; //Error no ReadList is registerd Request denied
             END_IF;
           END_IF;

           IF #tempReadTrigger THEN
             #statOpcUaRequests.Read := TRUE;
             #statBusy := TRUE;
             #statStatus := #STATUS_BUSY;
           ELSE
             #statOpcUaRequests.Read := FALSE;
           END_IF;
           //Error
           IF #instOpcUaReadList.Error THEN
             //--> Call ConnectionGetStatus if Status = "16#800D0000"
             IF #instOpcUaReadList.Status = #STATUS_SERVER_NOT_CONNECTED THEN
               #statCase := #CASE_CONNECTION_GET_STATUS;
             END_IF;
             #statOpcUaRequests.Read := FALSE;
             // => OUT
             #statError := TRUE;
             #statBusy := FALSE;
             #statStatus := #instOpcUaReadList.Status;
             #statErrorId := #ERR_ID_RL;
           END_IF;

           //Done
           IF #instOpcUaReadList.Done THEN
             //Check StatusList
             FOR #tempIndex := 0 TO UDINT_TO_INT(CountOfElements(#readNodeIds) - 1) DO
               IF #statOpcUaStatusLists.#ReadList[#tempIndex] <> 16#0 THEN
                 // => OUT
                 #statError := TRUE;
                 #statDone := FALSE;
                 #statBusy := FALSE;
                 #statStatus := #statOpcUaStatusLists.#ReadList[#tempIndex];
                 #statErrorId := #ERR_ID_RL;
                 EXIT;
               END_IF;
             END_FOR;
             #statOpcUaRequests.Read := FALSE;
             // => OUT
             IF NOT #statError THEN
               #statDone := TRUE;
               #statBusy := FALSE;
               #statError := FALSE;
               #statStatus := #STATUS_DONE;
               #statErrorId := #ERR_ID_GOOD;
               //Count up statReadCount
               #statReadCount += 1;
               //--> Nodes are read continously ...
             END_IF;
           END_IF;
         END_REGION

         REGION Write
           //Trigger
           IF #statRegisteredWrite THEN
             #instWriteTrigger(CLK := #write,
                               Q => #tempWriteTrigger);
           ELSE
             IF #write THEN
               #statError := TRUE;
               #statErrorId := #ERR_ID_WL;
               #statStatus := #STATUS_NOT_REGISTERED; //Error no WriteList is registerd Request denied
             ELSE
               #statError := FALSE;
               #statErrorId := #ERR_ID_GOOD;
               #statStatus := #STATUS_IDLE; //Error no WriteList is registerd Request denied
             END_IF;
           END_IF;

           IF #tempWriteTrigger THEN
             #statOpcUaRequests.Write := TRUE;
             #statBusy := TRUE;
             #statStatus := #STATUS_BUSY;
           ELSE
             #statOpcUaRequests.Write := FALSE;
           END_IF;
           //Error
           IF #instOpcUaWriteList.Error THEN
             //--> Call ConnectionGetStatus if Status = "16#800D0000"
             IF #instOpcUaWriteList.Status = #STATUS_SERVER_NOT_CONNECTED THEN
               #statCase := #CASE_CONNECTION_GET_STATUS;
             END_IF;
             #statOpcUaRequests.Write := FALSE;
             // => OUT
             #statError := TRUE;
             #statBusy := FALSE;
             #statStatus := #instOpcUaWriteList.Status;
             #statErrorId := #ERR_ID_WL;
           END_IF;

           //Done
           IF #instOpcUaWriteList.Done THEN
             //Check StatusList
             FOR #tempIndex := 0 TO UDINT_TO_INT(CountOfElements(#writeNodeIds) - 1) DO
               IF #statOpcUaStatusLists.#WriteList[#tempIndex] <> 16#0 THEN
                 // => OUT
                 #statError := TRUE;
                 #statDone := FALSE;
                 #statBusy := FALSE;
                 #statStatus := #statOpcUaStatusLists.#WriteList[#tempIndex];
                 #statErrorId := #ERR_ID_WL;
                 EXIT;
               END_IF;
             END_FOR;

             #statOpcUaRequests.Write := FALSE;
             // => OUT
             IF NOT #statError THEN
               #statDone := TRUE;
               #statBusy := FALSE;
               #statError := FALSE;
               #statStatus := #STATUS_DONE;
               #statErrorId := #ERR_ID_GOOD;
               //Count up statwriteCount
               #statWriteCount += 1;
               //--> Nodes are write continously ...
             END_IF;
           END_IF;
         END_REGION

         REGION Method Call
           //Trigger
           IF #statRegisteredMethods THEN
             #instMethodCallTrigger(CLK := #callMethod,
                                    Q => #tempMethodCallTrigger);
           ELSE
             IF #callMethod THEN
               #statError := TRUE;
               #statErrorId := #ERR_ID_MC;
               #statStatus := #STATUS_NOT_REGISTERED; //Error no MethodList is registerd Request denied
             ELSE
               #statError := FALSE;
               #statErrorId := #ERR_ID_GOOD;
               #statStatus := #STATUS_IDLE; //Error no MethodList is registerd Request denied
             END_IF;
           END_IF;

           IF #tempMethodCallTrigger THEN
             #statMethodHdlId := #methodHdlIndex * 0;
             //Define statMethodHdl for the input methodHdlIndex choosen index of MethodList
             #tempRetVal := Serialize(SRC_VARIABLE := #methodHdls,
                                      DEST_ARRAY => #statSerializeMethodHdls,
                                      POS := #statMethodHdlId);
             IF #tempRetVal <> 0 THEN
               #statErrorId := #ERR_ID_MC;
               #statStatus := 16#8000 + INT_TO_DWORD(#tempRetVal);
               #statError := TRUE;
             ELSE
               #statMethodHdlId := #methodHdlIndex * 4;
               #statMethodHdl.%B0 := #statSerializeMethodHdls[#statMethodHdlId + 3];
               #statMethodHdl.%B1 := #statSerializeMethodHdls[#statMethodHdlId + 2];
               #statMethodHdl.%B2 := #statSerializeMethodHdls[#statMethodHdlId + 1];
               #statMethodHdl.%B3 := #statSerializeMethodHdls[#statMethodHdlId];
               //Start Method Call
               #statOpcUaRequests.MethodCall := TRUE;
               #statBusy := TRUE;
               #statStatus := #STATUS_BUSY;
             END_IF;
           ELSE
             #statOpcUaRequests.MethodCall := FALSE;
           END_IF;
           //Error
           IF #instOpcUaMethodCall.Error THEN
             //--> Call ConnectionGetStatus if Status = "16#800D0000"
             IF #instOpcUaMethodCall.Status = #STATUS_SERVER_NOT_CONNECTED THEN
               #statCase := #CASE_CONNECTION_GET_STATUS;
             END_IF;
             #statOpcUaRequests.MethodCall := FALSE;
             // => OUT
             #statError := TRUE;
             #statBusy := FALSE;
             #statStatus := #instOpcUaMethodCall.Status;
             #statErrorId := #ERR_ID_MC;
           END_IF;

           //Done
           IF #instOpcUaMethodCall.Done THEN
             //Check MethodResult
             IF #statMethodResult <> 0 THEN
               #statError := TRUE;
               #statBusy := FALSE;
               #statStatus := #statMethodResult;
               #statErrorId := #ERR_ID_MC;
             END_IF;
             #statOpcUaRequests.MethodCall := FALSE;
             // => OUT
             #statDone := TRUE;
             #statBusy := FALSE;
             #statError := FALSE;
             #statStatus := #STATUS_DONE;
             #statErrorId := #ERR_ID_GOOD;
             //Count up statwriteCount
             #statMethodCallCount += 1;
             //--> Methods can be called continously ...
           END_IF;

         END_REGION

         REGION Clear Session 
           #instClearConnTrig(CLK := NOT #connect,
                              Q => #tempRHLTrigger);

           IF #tempRHLTrigger THEN
             #statRHLTrigger := TRUE;
             #statBusy := TRUE;
           END_IF;
           REGION Release lists
             //If Disconnect requested, release nodes -> disconnect established connection
             //-------DISCONNECT HANDLING------------
             //--------------------------------------
             IF #statRHLTrigger THEN
               IF #statRegisteredWrite AND #writeNodeIds <> NULL AND #writeNodeHdls <> NULL THEN
                 #statOpcUaRequests.RHLWrite := TRUE;
                 #statStatus := #STATUS_BUSY;
               ELSE
                 IF #statRegisteredRead AND #readNodeIds <> NULL AND #readNodeHdls <> NULL THEN
                   #statOpcUaRequests.RHLRead := TRUE;
                   #statStatus := #STATUS_BUSY;
                 ELSE
                   IF #statRegisteredMethods AND #methodNodeIds <> NULL AND #methodHdls <> NULL AND #objNodeIds <> NULL THEN
                     #statOpcUaRequests.RHLMethods := TRUE;
                     #statStatus := #STATUS_BUSY;
                   ELSE
                     #statRHLTrigger := FALSE;
                     #statStatus := #STATUS_IDLE;
                   END_IF;
                 END_IF;
               END_IF;
             END_IF;
             REGION Release ReadList
               //Release Handle List of Read Nodes was not successful
               IF #InstOpcUaRHLRead.Error THEN
                 //--> Call ConnectionGetStatus if Status = "16#800D0000"
                 IF #InstOpcUaRHLRead.Status = #STATUS_SERVER_NOT_CONNECTED THEN
                   #statCase := #CASE_CONNECTION_GET_STATUS;
                 END_IF;
                 #statOpcUaRequests.RHLRead := FALSE;
                 // => OUT
                 #statError := TRUE;
                 #statStatus := #InstOpcUaRHLRead.Status;
                 #statErrorId := #ERR_ID_R_RHL;
               END_IF;

               //Release Handle List of Read Nodes was successful
               IF #InstOpcUaRHLRead.Done THEN
                 //Check StatusList
                 FOR #tempIndex := 0 TO UDINT_TO_INT(CountOfElements(#readNodeIds) - 1) DO
                   IF #statOpcUaStatusLists.#ReadRHL[#tempIndex] <> 16#0 THEN
                     // => OUT
                     #statError := TRUE;
                     #statDone := FALSE;
                     #statBusy := FALSE;
                     #statStatus := #statOpcUaStatusLists.#ReadRHL[#tempIndex];
                     #statErrorId := #ERR_ID_R_RHL;
                     EXIT;
                   END_IF;
                 END_FOR;
                 #statOpcUaRequests.RHLRead := FALSE;
                 #statRegisteredRead := FALSE;
                 IF NOT #statError THEN
                   // => OUT
                   #statBusy := FALSE;
                   #statError := FALSE;
                   #statStatus := #STATUS_DONE;
                   #statErrorId := #ERR_ID_GOOD;
                   //--> Nodes are released
                 END_IF;
               END_IF;
             END_REGION

             REGION Release WriteList
               //Release Handle List of Write Nodes was not successful
               IF #instOpcUaRHLWrite.Error THEN
                 //--> Call ConnectionGetStatus if Status = "16#800D0000"
                 IF #instOpcUaRHLWrite.Status = #STATUS_SERVER_NOT_CONNECTED THEN
                   #statCase := #CASE_CONNECTION_GET_STATUS;
                 END_IF;
                 #statOpcUaRequests.RHLWrite := FALSE;
                 // => OUT
                 #statError := TRUE;
                 #statStatus := #instOpcUaRHLWrite.Status;
                 #statErrorId := #ERR_ID_W_RHL;
               END_IF;

               //Release Handle List of Write Nodes was successful
               IF #instOpcUaRHLWrite.Done THEN
                 //Check StatusList
                 FOR #tempIndex := 0 TO UDINT_TO_INT(CountOfElements(#writeNodeIds) - 1) DO
                   IF #statOpcUaStatusLists.WriteRHL[#tempIndex] <> 16#0 THEN
                     // => OUT
                     #statError := TRUE;
                     #statDone := FALSE;
                     #statBusy := FALSE;
                     #statStatus := #statOpcUaStatusLists.#WriteRHL[#tempIndex];
                     #statErrorId := #ERR_ID_W_RHL;
                     EXIT;
                   END_IF;
                 END_FOR;
                 #statOpcUaRequests.RHLWrite := FALSE;
                 #statRegisteredWrite := FALSE;
                 IF NOT #statError THEN
                   // => OUT
                   #statBusy := FALSE;
                   #statError := FALSE;
                   #statStatus := #STATUS_DONE;
                   #statErrorId := #ERR_ID_GOOD;
                   //--> Nodes are released
                 END_IF;
               END_IF;
             END_REGION

             REGION Release MethodList
               //Release Handle List of Methods was not successful
               IF #instOpcUaRHLMethods.Error THEN
                 //--> Call ConnectionGetStatus if Status = "16#800D0000"
                 IF #instOpcUaRHLMethods.Status = #STATUS_SERVER_NOT_CONNECTED THEN
                   #statCase := #CASE_CONNECTION_GET_STATUS;
                 END_IF;
                 #statOpcUaRequests.RHLMethods := FALSE;
                 // => OUT
                 #statError := TRUE;
                 #statStatus := #instOpcUaRHLMethods.Status;
                 #statErrorId := #ERR_ID_M_RHL;
               END_IF;

               //Release Handle List of Methods was successful
               IF #instOpcUaRHLMethods.Done THEN
                 //Check StatusList
                 FOR #tempIndex := 0 TO UDINT_TO_INT(CountOfElements(#methodNodeIds) - 1) DO
                   IF #statOpcUaStatusLists.#MethodRHL[#tempIndex] <> 16#0 THEN
                     // => OUT
                     #statError := TRUE;
                     #statDone := FALSE;
                     #statBusy := FALSE;
                     #statStatus := #statOpcUaStatusLists.#MethodRHL[#tempIndex];
                     #statErrorId := #ERR_ID_M_RHL;
                     EXIT;
                   END_IF;
                 END_FOR;
                 #statOpcUaRequests.RHLMethods := FALSE;
                 #statRegisteredMethods := FALSE;
                 IF NOT #statError THEN
                   // => OUT
                   #statBusy := FALSE;
                   #statError := FALSE;
                   #statStatus := #STATUS_DONE;
                   #statErrorId := #ERR_ID_GOOD;
                   //--> Nodes are released
                 END_IF;
               END_IF;
             END_REGION
           END_REGION

           REGION Disconnect
             #instDisconRTrig(CLK := NOT #statRegisteredRead
                              AND NOT #statRegisteredWrite
                              AND NOT #statRegisteredMethods,
                              //OR (#statConnected AND #statErrorId > 70),
                              Q => #tempDisconnectTrigger);

             IF #tempDisconnectTrigger THEN
               IF #statConnectionHdl <> 16#0 THEN
                 #statOpcUaRequests.Disconnect := TRUE;
                 //set FB Outputs
                 #statBusy := TRUE;
                 #statStatus := #STATUS_BUSY;
                 #statConnectionHdl := 0;
               ELSE
                 #statCase := #CASE_CONNECT;
                 //Error No connection established
               END_IF;
             ELSE
               #statOpcUaRequests.Disconnect := FALSE;
             END_IF;

             //Error at connection establishment
             IF #instOpcUaDisconnect.Error THEN
               #statError := TRUE;
               #statBusy := FALSE;
               #statErrorId := #ERR_ID_DISCON;
               #statStatus := #instOpcUaDisconnect.Status;
               #statCase := #CASE_CONNECTION_GET_STATUS;
             END_IF;

             //Disconnect was successful
             IF #instOpcUaDisconnect.Done THEN
               #statConnected := FALSE;
               #statDone := FALSE;
               #statNamespaceIndexesSet := FALSE;
               #statBusy := FALSE;
               #statOpcUaRequests.Disconnect := FALSE;
               IF #statErrorId <> 0 THEN
                 #statError := TRUE;
               ELSE
                 #statError := FALSE;
                 #statErrorId := #ERR_ID_GOOD;
                 #statStatus := #STATUS_DONE;
               END_IF;
               #statCase := #CASE_CONNECT;
             END_IF;
           END_REGION
         END_REGION
       END_REGION

     #CASE_CONNECTION_GET_STATUS:
       REGION Connection Diagnostics
         #statOpcUaRequests.ConGS := TRUE;
         IF #instOpcUaConnectionGetStatus.Error THEN
           //--> New connection attempt if Status "16#A0000105" (Session could not be reactivated and all resources are cleaned up)
           //or Status "16#80AE_0000" (The network connectoin hs been closed)
           IF #instOpcUaConnectionGetStatus.Status = #STATUS_SESSION_CLEANEDUP OR
             #instOpcUaConnectionGetStatus.Status = #STATUS_BAD_CONNECTION_CLOSED
           THEN
             //Connection is cleaned up
             #statConnected := FALSE;
             #statNamespaceIndexesSet := FALSE; //Namespace Indexes are set via OPC_UA_NamespaceGetIndexList
             #statRegisteredRead := FALSE; //Nodes are not registerd anymore
             #statRegisteredWrite := FALSE; //Nodes are not registerd anymore 
             #statRegisteredMethods := FALSE; //Nodes are not registerd anymore
             //Next Step --> New connection attempt
             #statCase := #CASE_CONNECT;
           END_IF;
           #statOpcUaRequests.ConGS := FALSE;
           // => OUT
           #statError := TRUE;
           #statBusy := FALSE;
           #statStatus := #instOpcUaConnectionGetStatus.Status;
           #statErrorId := #ERR_ID_CON_GS_STATUS;
         END_IF;
         //Done
         IF #instOpcUaConnectionGetStatus.Done THEN
           //ConnectionStatus+ServerState+ServiceLevel are "Good"
           IF #instOpcUaConnectionGetStatus.ConnectionStatus = #UACS_CONNECTED
             AND #instOpcUaConnectionGetStatus.ServerState = #UASS_RUNNING
             AND #instOpcUaConnectionGetStatus.ServiceLevel = #UASL_GOOD
           THEN
             #statOpcUaRequests.ConGS := FALSE;
             //Session is reactivated and nodes are still registered --> Next Step --> CommandAndIdle
             IF #statConnected AND #statNamespaceIndexesSet
               AND (#statRegisteredRead OR #readNodeIds = NULL)
               AND (#statRegisteredWrite OR #writeNodeIds = NULL)
               AND (#statRegisteredMethods OR #methodNodeIds = NULL)
             THEN
               #statBusy := FALSE;
               #statCase := #CASE_CONNECTED;
               //Session is reactivated and nodes are not registered yet --> Next Step --> NodeGetHandleList
             ELSIF #statConnected AND #statNamespaceIndexesSet
               AND (NOT #statRegisteredRead OR NOT #statRegisteredWrite OR NOT #statRegisteredMethods)
             THEN
               #statCase := #CASE_NODE_GET_HANDLE_LIST;
               //Session is reactivated and namespaceIndexes are not set yet --> Next Step --> NamespaceGetIndexList
             ELSIF #statConnected AND NOT #statNamespaceIndexesSet
               AND (NOT #statRegisteredRead OR NOT #statRegisteredWrite OR NOT #statRegisteredMethods)
             THEN
               #statCase := #CASE_NAMESPACE_GET_INDEX_LIST;
               //Session is reactivated (but connected bit isn't set) and namespaceIndexes are set and nodes are registered
               //--> Next Step --> CommandAndIdle
             ELSIF NOT #statConnected AND #statNamespaceIndexesSet
               AND (#statRegisteredRead OR #readNodeIds = NULL)
               AND (#statRegisteredWrite OR #writeNodeIds = NULL)
               AND (#statRegisteredMethods OR #methodNodeIds = NULL)
             THEN
               //connected has to be set
               #statConnected := TRUE;
               #statBusy := FALSE;
               #statRHLTrigger := FALSE;
               #statOpcUaRequests.RHLWrite := FALSE;
               #statOpcUaRequests.RHLRead := FALSE;
               #statOpcUaRequests.RHLMethods := FALSE;
               #statCase := #CASE_CONNECTED;
             END_IF;
           ELSE
             IF #connect THEN
               //ConnectionStatus is not "Good"
               IF #instOpcUaConnectionGetStatus.ConnectionStatus <> #UACS_CONNECTED THEN
                 #statOpcUaRequests.ConGS := FALSE;
                 // => OUT
                 #statError := TRUE;
                 #statBusy := FALSE;
                 #statConnected := FALSE;
                 #statErrorId := #ERR_ID_CON_GS_CSTATE;
                 #statStatus := #instOpcUaConnectionGetStatus.ConnectionStatus;
                 //ServerState is not "Good"
               ELSIF #instOpcUaConnectionGetStatus.ServerState <> #UASS_RUNNING THEN
                 #statOpcUaRequests.ConGS := FALSE;
                 // => OUT
                 #statError := TRUE;
                 #statBusy := FALSE;
                 #statConnected := FALSE;
                 #statStatus := #instOpcUaConnectionGetStatus.ServerState;
                 #statErrorId := #ERR_ID_CON_GS_SSTATE;
                 //ServiceLevel is not "Good"
               ELSIF #instOpcUaConnectionGetStatus.ServiceLevel <> #UASL_GOOD THEN
                 #statOpcUaRequests.ConGS := FALSE;
                 // => OUT
                 #statError := TRUE;
                 #statBusy := FALSE;
                 #statStatus := #instOpcUaConnectionGetStatus.ServiceLevel;
                 #statErrorId := #ERR_ID_CON_GS_SLVL;
               END_IF;
             ELSE
               //connect is not set -> connection was faulty -> back to case CONNECT
               //new connection can be set up
               #statCase := #CASE_CONNECT;
               #statOpcUaRequests.ConGS := FALSE;
               #statRHLTrigger := FALSE;
               #statNamespaceIndexesSet := FALSE;
               #statRegisteredRead := FALSE;
               #statRegisteredWrite := FALSE;
               #statRegisteredMethods := FALSE;
             END_IF;
           END_IF;
         END_IF;
       END_REGION
     ELSE  // Statement section ELSE
       ; //Not reachable
   END_CASE;

   REGION Call SFBs
     //CALL SFB OPC_UA_Connect
     #instOpcUaConnect(REQ := #statOpcUaRequests.Connect,
                       ServerEndpointUrl := #serverEndpointUrl,
                       SessionConnectInfo := #connectionInfo,
                       Timeout := #OPC_UA_FUNCTIONS_TIMEOUT,
                       ConnectionHdl => #statConnectionHdl);

     //CALL SFB OPC_UA_NamespaceGetIndexList 
     #instOpcUaNamespaceGIL(REQ := #statOpcUaRequests.NGIL,
                            ConnectionHdl := #statConnectionHdl,
                            NamespaceUrisCount := UDINT_TO_UINT(CountOfElements(#namespaceUris)),
                            NamespaceUris := #namespaceUris,
                            Timeout := #OPC_UA_FUNCTIONS_TIMEOUT,
                            StatusList := #statOpcUaStatusLists.#NamespaceGIL,
                            NamespaceIndexes := #namespaceIndexes);

     //CALL SFB OPC_UA_NodeGetHandleList_Read
     #InstOpcUaGHLRead(REQ := #statOpcUaRequests.GHLRead,
                       ConnectionHdl := #statConnectionHdl,
                       NodeIDCount := UDINT_TO_UINT(CountOfElements(#readNodeIds)),
                       NodeIDs := #readNodeIds,
                       Timeout := #OPC_UA_FUNCTIONS_TIMEOUT,
                       NamespaceIndexCount := UDINT_TO_UINT(CountOfElements(#namespaceIndexes)),
                       NamespaceIndexes := #namespaceIndexes,
                       NodeStatusList := #statOpcUaStatusLists.#ReadGHL,
                       NodeHdls := #readNodeHdls);

     //CALL SFB OPC_UA_NodeGetHandleList_Write
     #instOpcUaGHLWrite(REQ := #statOpcUaRequests.GHLWrite,
                        ConnectionHdl := #statConnectionHdl,
                        NodeIDCount := UDINT_TO_UINT(CountOfElements(#writeNodeIds)),
                        NodeIDs := #writeNodeIds,
                        Timeout := #OPC_UA_FUNCTIONS_TIMEOUT,
                        NamespaceIndexCount := UDINT_TO_UINT(CountOfElements(#namespaceIndexes)),
                        NamespaceIndexes := #namespaceIndexes,
                        NodeStatusList := #statOpcUaStatusLists.#WriteGHL,
                        NodeHdls := #writeNodeHdls);

     //CALL SFB OPC_UA_MethodGetHandleList
     #instOpcUaGHLMethods(REQ := #statOpcUaRequests.GHLMethods,
                          ConnectionHdl := #statConnectionHdl,
                          NodeIDCount := UDINT_TO_UINT(CountOfElements(#methodNodeIds)),
                          ObjectNodeIDs := #objNodeIds,
                          MethodNodeIDs := #methodNodeIds,
                          Timeout := #OPC_UA_FUNCTIONS_TIMEOUT,
                          NamespaceIndexCount := UDINT_TO_UINT(CountOfElements(#namespaceIndexes)),
                          NamespaceIndexes := #namespaceIndexes,
                          StatusList := #statOpcUaStatusLists.#MethodGHL,
                          MethodHdls := #methodHdls);

     //CALL SFB OPC_UA_ReadList
     #instOpcUaReadList(REQ := #statOpcUaRequests.Read,
                        ConnectionHdl := #statConnectionHdl,
                        NodeHdlCount := UDINT_TO_UINT(CountOfElements(#readNodeHdls)),
                        NodeHdls := #readNodeHdls,
                        Timeout := #OPC_UA_FUNCTIONS_TIMEOUT,
                        NodeStatusList := #statOpcUaStatusLists.#ReadList,
                        TimeStamps := #statOpcUaReadTimeStamps,
                        Variable := #readData);

     //CALL SFB OPC_UA_WriteList
     #instOpcUaWriteList(REQ := #statOpcUaRequests.Write,
                         ConnectionHdl := #statConnectionHdl,
                         NodeHdlCount := UDINT_TO_UINT(CountOfElements(#writeNodeHdls)),
                         NodeHdls := #writeNodeHdls,
                         Timeout := #OPC_UA_FUNCTIONS_TIMEOUT,
                         NodeStatusList := #statOpcUaStatusLists.#WriteList,
                         Variable := #writeData);

     //CALL SFB OPC_UA_MethodCall
     #instOpcUaMethodCall(REQ := #statOpcUaRequests.MethodCall,
                          ConnectionHdl := #statConnectionHdl,
                          MethodHdl := #statMethodHdl,
                          Timeout := #OPC_UA_FUNCTIONS_TIMEOUT,
                          MethodResult := #statMethodResult,
                          InputArguments := #inputArguments,
                          OutputArguments := #outputArguments);

     //CALL SFB OPC_UA_NodeReleaseHandleList_Read
     #InstOpcUaRHLRead(REQ := #statOpcUaRequests.RHLRead,
                       ConnectionHdl := #statConnectionHdl,
                       NodeHdlCount := UDINT_TO_UINT(CountOfElements(#readNodeHdls)),
                       NodeHdls := #readNodeHdls,
                       Timeout := #OPC_UA_FUNCTIONS_TIMEOUT,
                       NodeStatusList := #statOpcUaStatusLists.#ReadRHL);

     //CALL SFB OPC_UA_NodeReleaseHandleList_Write
     #instOpcUaRHLWrite(REQ := #statOpcUaRequests.RHLWrite,
                        ConnectionHdl := #statConnectionHdl,
                        NodeHdlCount := UDINT_TO_UINT(CountOfElements(#writeNodeHdls)),
                        NodeHdls := #writeNodeHdls,
                        Timeout := #OPC_UA_FUNCTIONS_TIMEOUT,
                        NodeStatusList := #statOpcUaStatusLists.#WriteRHL);

     //CALL SFB OPC_UA_MethodReleaseHandleList
     #instOpcUaRHLMethods(REQ := #statOpcUaRequests.RHLMethods,
                          ConnectionHdl := #statConnectionHdl,
                          MethodHdlCount := UDINT_TO_UINT(CountOfElements(#methodHdls)),
                          MethodHdls := #methodHdls,
                          Timeout := #OPC_UA_FUNCTIONS_TIMEOUT,
                          StatusList := #statOpcUaStatusLists.#MethodRHL);

     //CALL SFB OPC_UA_Disconnect
     #instOpcUaDisconnect(REQ := #statOpcUaRequests.Disconnect,
                          ConnectionHdl := #statConnectionHdl,
                          Timeout := #OPC_UA_FUNCTIONS_TIMEOUT);

     //CALL SFB OPC_UA_ConnectionGetStatus
     #instOpcUaConnectionGetStatus(REQ := #statOpcUaRequests.ConGS,
                                   ConnectionHdl := #statConnectionHdl,
                                   Timeout := #OPC_UA_FUNCTIONS_TIMEOUT);
   END_REGION

   REGION Set FB Outputs
     #connected := #statConnected;
     #done := #statDone;
     #busy := #statBusy;
     #errorId := #statErrorId;
     #error := #statError;
     #status := #statStatus;
     #conectionHdl := #statConnectionHdl;
   END_REGION
END_FUNCTION_BLOCK